(* This function Block interfaces with a NO turbo valve*)
(* Mainly used in the FEE HXR GATT*)
FUNCTION F_TurboExtILK_NO : BOOL
VAR_INPUT
    Turbo		:	ST_PTM;
    BackingGauge:	ST_VG;
    InletGauge	:	ST_VG;
    VentValve	:	ST_VCC_NO; //NO type turbo valve
    ScrollPump	:	ST_RoughPump;
END_VAR

VAR
END_VAR

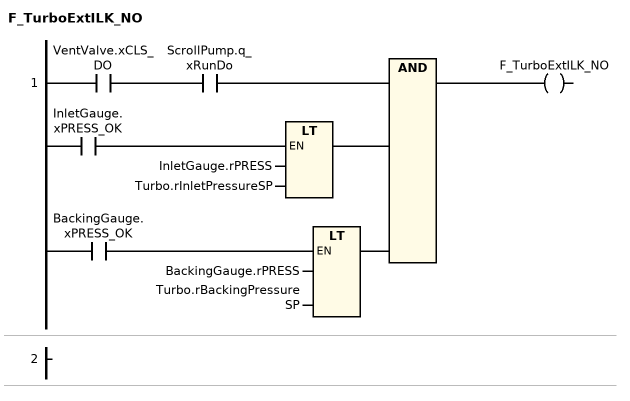
// NETWORK 1
F_TurboExtILK_NO := (VentValve.xCLS_DO AND ScrollPump.q_xRunDo) AND (InletGauge.xPRESS_OK AND InletGauge.rPRESS < Turbo.rInletPressureSP) AND (BackingGauge.xPRESS_OK AND BackingGauge.rPRESS < Turbo.rBackingPressureSP);

// NETWORK 2

END_FUNCTION

(* stored: Version 1.1.0.1
   POU F_TurboExtILK_NO: Id {3f22491e-9c00-45b3-979a-0a023cc045c2}, SpecialFunc None *)
